FUNCTION_BLOCK Sensor_StateOrder_View
  (* Version 0.1, 2005-12-15, Oscar Ljungkrantz, Chalmers *)
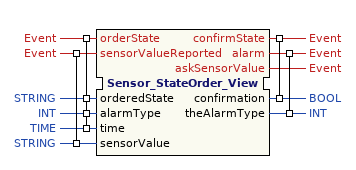
  EVENT_INPUT
    orderState WITH orderedState, alarmType, time;
    sensorValueReported WITH sensorValue;
  END_EVENT
  EVENT_OUTPUT
    confirmState WITH confirmation;
    alarm WITH theAlarmType;
    askSensorValue;
  END_EVENT
  VAR_INPUT
    orderedState : STRING;
    alarmType : INT;
    time : TIME;
    sensorValue : STRING;
  END_VAR
  VAR_OUTPUT
    confirmation : BOOL;
    theAlarmType : INT;
  END_VAR
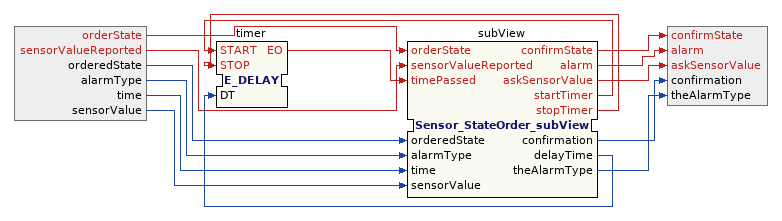
  FBS
    timer : E_DELAY;
    subView : Sensor_StateOrder_subView;
  END_FBS
  EVENT_CONNECTIONS
    orderState TO subView.orderState;
    sensorValueReported TO subView.sensorValueReported;
    subView.confirmState TO confirmState;
    subView.askSensorValue TO askSensorValue;
    subView.alarm TO alarm;
    subView.startTimer TO timer.START;
    subView.stopTimer TO timer.STOP;
    timer.EO TO subView.timePassed;
  END_CONNECTIONS
  DATA_CONNECTIONS
    orderedState TO subView.orderedState;
    alarmType TO subView.alarmType;
    time TO subView.time;
    sensorValue TO subView.sensorValue;
    subView.confirmation TO confirmation;
    subView.theAlarmType TO theAlarmType;
    subView.delayTime TO timer.DT;
  END_CONNECTIONS
END_FUNCTION_BLOCK
(* other elements stored in the file *)
(* Connections from this View to subView *)
(* Connections from subView to this View *)
(* Connections from subView to timer *)
(* Connections from timer to subView *)
(* Connections from this View to subView *)
(* Connections from subView to this View *)
(* Connections from subView to timer *)
